(* Logix 5000 project; controller Sucrose_Main Emulate 5570 rev 20.12; software revision 20.01 *)

TASK _00_Master (continuous, watchdog 500 ms) : Master_Main
TASK _01_Sucrose (event, rate 10 ms, priority 10, watchdog 500 ms) : CIP_RemoteArea_AutoLogic, CIP_RemoteArea_EN2T_IO_Discrete_DO_E20_4, CIP_RemoteArea_EN2T_IO_Discrete_DO_E20_5, CIP_RemoteArea_EN2T_IO_Discrete_DO_E20_6, CIP_RemoteArea_EN2T_IO_Discrete_DO_E24_1, CIP_RemoteArea_EN2T_IO_Discrete_DO_E24_2, CIP_RemoteArea_EN2T_IO_Discrete_DO_E25_4, CIP_RemoteArea_EN2T_IO_Discrete_DO_E25_5, CIP_RemoteArea_EN2T_IO_Drives, DischargeArea_AutoLogic, DischargeArea_EN2T_IO_Discrete_DO_E20_3, DischargeArea_EN2T_IO_Discrete_DO_E20_4, DischargeArea_EN2T_IO_Discrete_DO_E20_5, DischargeArea_EN2T_IO_Discrete_DO_E20_6, DischargeArea_EN2T_IO_Discrete_DO_E20_7, DischargeArea_EN2T_IO_Discrete_DO_E24_3, DischargeArea_EN2T_IO_Drives, FiltrationArea_AutoLogic, FiltrationArea_EN2T_IO_Discrete_DO_E22_2, FiltrationArea_EN2T_IO_Discrete_DO_E22_3, FiltrationArea_EN2T_IO_Discrete_DO_E22_4

MODULES
   Local : Emulate 5570 (ICP 5, rev 20.12)
      EN2T_CCN : 1756-EN2T (ICP 1, Ethernet 192.168.15.49, rev 10.1)
      EN2T_IO : 1756-EN2T (ICP 2, Ethernet 192.168.1.1, rev 10.1)
         P620101 : PowerFlex 525-EENET (Ethernet 192.168.1.32, rev 3.1, Output RPI 20 ms)
         P230010 : PowerFlex 525-EENET (Ethernet 192.168.1.33, rev 4.1, Output RPI 20 ms)
         P230401 : PowerFlex 525-EENET (Ethernet 192.168.1.30, rev 2.2, Output RPI 20 ms)
         P230020 : PowerFlex 525-EENET (Ethernet 192.168.1.34, rev 4.1, Output RPI 20 ms)
         P230402 : PowerFlex 525-EENET (Ethernet 192.168.1.31, rev 4.1, Output RPI 20 ms)
         FLX_E25 : 1794-AENT (Ethernet 192.168.1.25, rev 4.1, Output RPI 20 ms)
            FLX_E25_2 : 1794-IB16 (Flex 2, rev 1.1)
            FLX_E25_5 : vendor 1 type 7 code 45 (Flex 5, rev 1.1)
            FLX_E25_4 : vendor 1 type 7 code 45 (Flex 4, rev 1.1)
            FLX_E25_3 : 1794-IB16 (Flex 3, rev 1.1)
            FLX_E25_1 : 1794-VHSC (Flex 1, rev 1.1, Output RPI 50 ms)
            FLX_E25_0 : vendor 1 type 10 code 25 (Flex 0, rev 2.1, Input RPI 80 ms)
         FLX_E20 : 1794-AENT (Ethernet 192.168.1.20, rev 4.1, Output RPI 20 ms)
            FLX_E20_7 : 1794-OW8 (Flex 7, rev 1.1)
            FLX_E20_4 : vendor 1 type 7 code 45 (Flex 4, rev 1.1)
            FLX_E20_5 : vendor 1 type 7 code 45 (Flex 5, rev 1.1)
            FLX_E20_1 : 1794-IB16 (Flex 1, rev 1.1)
            FLX_E20_6 : vendor 1 type 7 code 45 (Flex 6, rev 1.1)
            FLX_E20_2 : 1794-IB16 (Flex 2, rev 1.1)
            FLX_E20_0 : 1794-IB16 (Flex 0, rev 1.1)
            FLX_E20_3 : vendor 1 type 7 code 45 (Flex 3, rev 1.1)
         FLX_E24 : 1794-AENT (Ethernet 192.168.1.24, rev 4.1, Output RPI 20 ms)
            FLX_E24_5 : 1794-OW8 (Flex 5, rev 1.1)
            FLX_E24_0 : vendor 1 type 7 code 45 (Flex 0, rev 1.1)
            FLX_E24_4 : vendor 1 type 7 code 45 (Flex 4, rev 1.1)
            FLX_E24_1 : vendor 1 type 7 code 45 (Flex 1, rev 1.1)
            FLX_E24_2 : vendor 1 type 7 code 45 (Flex 2, rev 1.1)
            FLX_E24_3 : vendor 1 type 7 code 45 (Flex 3, rev 1.1)
            FLX_E24_6 : 1794-OW8 (Flex 6, rev 1.1)
         FLX_E21 : 1794-AENT (Ethernet 192.168.1.21, rev 4.1, Output RPI 20 ms)
            FLX_E21_1 : vendor 1 type 10 code 25 (Flex 1, rev 2.1, Input RPI 80 ms)
            FLX_E21_2 : vendor 1 type 10 code 25 (Flex 2, rev 2.1, Input RPI 80 ms)
            FLX_E21_0 : vendor 1 type 10 code 25 (Flex 0, rev 2.1, Input RPI 80 ms)
         FLX_E23 : 1794-AENT (Ethernet 192.168.1.23, rev 4.1, Output RPI 20 ms)
            FLX_E23_6 : 1794-IB16 (Flex 6, rev 1.1)
            FLX_E23_5 : 1794-IB16 (Flex 5, rev 1.1)
            FLX_E23_4 : 1794-IB16 (Flex 4, rev 1.1)
            FLX_E23_3 : 1794-IB16 (Flex 3, rev 1.1)
            FLX_E23_0 : vendor 1 type 10 code 25 (Flex 0, rev 2.1, Input RPI 80 ms)
            FLX_E23_2 : vendor 1 type 10 code 25 (Flex 2, rev 2.1, Input RPI 80 ms)
            FLX_E23_1 : vendor 1 type 10 code 25 (Flex 1, rev 2.1, Input RPI 80 ms)
         FLX_E22 : 1794-AENT (Ethernet 192.168.1.22, rev 4.1, Output RPI 20 ms)
            FLX_E22_2 : vendor 1 type 7 code 45 (Flex 2, rev 1.1)
            FLX_E22_7 : vendor 1 type 7 code 45 (Flex 7, rev 1.1)
            FLX_E22_5 : vendor 1 type 7 code 45 (Flex 5, rev 1.1)
            FLX_E22_1 : 1794-IB16 (Flex 1, rev 1.1)
            FLX_E22_4 : vendor 1 type 7 code 45 (Flex 4, rev 1.1)
            FLX_E22_0 : 1794-IB16 (Flex 0, rev 1.1)
            FLX_E22_3 : vendor 1 type 7 code 45 (Flex 3, rev 1.1)
            FLX_E22_6 : vendor 1 type 7 code 45 (Flex 6, rev 1.1)
END_MODULES

TYPE Area_Ladder :
STRUCT
   BIT_Comment : BOOL;   // For Rung Comment
   BIT_Alarm : DINT[1];   // For Logic Alarms
   BIT_ONS : BOOL[32];   // For Logic One Shot Bits
   TMR_Alarm : TIMER[25];   // For Logic Alarm Timers
   BIT_Logic : DINT[5];   // For Logic Bits
   SP_Logic : DINT[10];   // For Logic Setpoints
   TMR_Logic : TIMER[10];   // For Logic Timers
   CTR_Logic : COUNTER[5];   // For Logic Counters
   CALC_Logic : REAL[10];   // For Logic Math Calculations
   STRING_Logic : STRING[5];   // For Logic Strings
   BIT_HMI : DINT[10];   // For HMI Buttons
   SP_HMI : DINT[10];   // For HMI Setpoints
   STATUS_HMI : DINT[10];   // For HMI Display Words
   STATUS_BIT_HMI : DINT[10];   // For HMI Display Bits
   STRING_HMI : STRING[5];   // For HMI Strings
END_STRUCT
END_TYPE

TYPE Area_Program :
STRUCT
   BIT_Comment : BOOL;   // For Rung Comment
   BIT_Alarm : DINT[2];   // For Logic Alarms
   BIT_ONS : BOOL[128];   // For Logic One Shot Bits
   TMR_Alarm : TIMER[50];   // For Logic Alarm Timers
   BIT_Logic : DINT[10];   // For Logic Bits
   SP_Logic : DINT[25];   // For Logic Setpoints
   TMR_Logic : TIMER[50];   // For Logic Timers
   CTR_Logic : COUNTER[10];   // For Logic Counters
   CALC_Logic : REAL[25];   // For Logic Math Calculations
   STRING_Logic : STRING[5];   // For Logic Strings
   BIT_HMI : DINT[10];   // For HMI Buttons
   SP_HMI : DINT[25];   // For HMI Setpoints
   STATUS_HMI : DINT[10];   // For HMI Display Words
   STATUS_BIT_HMI : DINT[10];   // For HMI Display Bits
   STRING_HMI : STRING[5];   // For HMI Strings
   TMR_Debounce_On : TIMER[50];   // For Inputs Debounce Timer On
   TMR_Debounce_Off : TIMER[50];   // For Inputs Debounce Timer Off
END_STRUCT
END_TYPE

TYPE CIP_CURRENT_FUNCTIONS_REMOTE :
STRUCT
   F1 : DINT;   // CIP FUNCTION 1
   StepDescription : STRING;   // CIP STRING
   TIME : INT;   // CIP STEP TIME
   VALID : DINT;   // CIP VALID STEP CONFIRMATION
   F2 : DINT;   // CIP FUNCTION 1
   F3 : DINT;   // CIP FUNCTION 1
END_STRUCT
END_TYPE

TYPE CIP_MASTER_FUNCTIONS_REMOTE :
STRUCT
   F1 : DINT[130];   // CIP FUNCTION 1
   StepDescription : STRING[130];   // CIP STRING
   TIME : INT[130];   // CIP STEP TIME
   F2 : DINT[130];   // CIP FUNCTION 1
   F3 : DINT[130];   // CIP FUNCTION 1
END_STRUCT
END_TYPE

TYPE CIP_REMOTE :
STRUCT
   STEP : DINT;   // CIP STEP NUMBER
   STATES : CIP_STATES_REMOTE;
   STEP_TIMER : TIMER;   // CIP STEP TIMER
   CURRENT : CIP_CURRENT_FUNCTIONS_REMOTE;   // CIP CURRENT FUNCTIONS
   MASTER : CIP_MASTER_FUNCTIONS_REMOTE;   // CIP SETPOINTS
   BIT_ONS : BOOL[32];   // REMOTE ONE SHOTS
   Selected : BOOL;   // CIP CIRCUIT SELECTED
END_STRUCT
END_TYPE

TYPE CIP_STATES_REMOTE :
STRUCT
   RUNNING : BOOL;   // CIP RUNNING BIT
   PAUSED : BOOL;   // CIP PAUSED BIT
   HOLDING : BOOL;   // CIP HOLDING BIT
   COMPLETE : BOOL;   // CIP COMPLETE BIT
   STEP_DONE : BOOL;   // CIP STEP DONE BIT
   GOOD_MOVE : BOOL;   // CIP GOOD MOVE BIT
   VALID : DINT;   // CIP VALID STEP WORK
   TIMER_ENABLE : BOOL;   // CIP TIMER ENABLE
END_STRUCT
END_TYPE

TYPE Date_Time :
STRUCT
   Year : DINT;
   Month : DINT;
   Day : DINT;
   Hour : DINT;
   Minute : DINT;
   Second : DINT;
   Millisecond : DINT;
END_STRUCT
END_TYPE

TYPE User_Login :
STRUCT
   User_Data : STRING[20];
   Password_Data : STRING[20];
   User_Input : STRING;
   Password_Input : STRING;
   Password_Level : DINT;
   Current_User : STRING;
   Blank_User : STRING;
   Blank_Password : STRING;
   Default_User : STRING;
   Clear_User : BOOL;
   Logout_PB : BOOL;
   Good_User : BOOL;
   Login_PB : BOOL;
END_STRUCT
END_TYPE

ADD_ON_INSTRUCTION PF525_VFD_E_ENET   (* revision 2.0 Deluxe Edition, vendor Eric Casciaro *)
// QSI Typical Logic for VFD Controlled Motor
// Revision note:
// AOI Revisions After Multiple Startups:
// Added PID Execute Logic
// Added Manual On Reset Logic During Alarm
// Added Zone & Device Specific Alarm Ack Logic
// Added Zone & Device Specific Clear Fault Logic
// Added Zone Manual Mode Enable Logic
// Added Speed Display Units Option Logic
// Added Device Overspeed Option Logic
// Added HMI Popup Display Options Configuration
VAR_IN_OUT
   PF525_In : AB:PowerFlex525V_E_ED09CCB8:I:0; {required}
   PF525_Out : AB:PowerFlex525V_EENET_Drive:O:0; {required}
END_VAR
VAR_INPUT
   ALM_ACK : BOOL; {required}   // Zone Master Alarm Acknowledge
   MM_Enable : BOOL; {required}   // Zone Master Manual Mode Enable
   CLR_Fault : BOOL; {required}   // Zone Master Clear Fault Enable
   Config_TMR_On_Preset : DINT; {visible}   // Configure Delay Start Timer Preset
   Config_TMR_Off_Preset : DINT; {visible}   // Configure Delay Stop Timer Preset
   Config_TMR_Alm_Preset : DINT; {visible}   // Configure Device Alarm Timer Preset
   Config_MO_ALM_Reset : BOOL;   // Configure Whether .MO Bit Turns Off After Alarm Condition
END_VAR
VAR_OUTPUT
   Config_Drive_Overspeed : BOOL; {access Read Only}   // Configure Whether the Drive Max Speed is Oversped (0 = 100 % or 60 Hz) (1 = 200% or 120 Hz)
   Config_HMI_Units_SpeedFeedback : BOOL;   // Configure Whether Speed Feedback is Shown in % or Hertz (0=%) (1=Hz)
   Config_HMI_Control_Reverse : BOOL;   // Configure Whether HMI Popup Allows Reverse Control
   Config_HMI_Control_Jog : BOOL;   // Configure Whether HMI Popup Allows Jog Control
END_VAR
VAR_INPUT
   Config_AS1 : BOOL;   // Configure Usage of Auto Speed 1
   Config_AS2 : BOOL;   // Configure Usage of Auto Speed 2
   Config_AS3 : BOOL;   // Configure Usage of Auto Speed 3
   Config_AS4 : BOOL;   // Configure Usage of Auto Speed 4
   Config_AS5 : BOOL;   // Configure Usage of Auto Speed 5
   Config_PID : BOOL; {visible}   // Configure Usage of PID Loop
   Config_PID_Kp : REAL;   // Configure PID Proportional Gain
   Config_PID_Ki : REAL;   // Configure PID Integral Gain
   Config_PID_Kd : REAL;   // Configure PID Derivative Gain
   SP_AS1 : DINT;   // Auto Speed Setpoint
   SP_AS2 : DINT;   // Auto Speed #2 Setpoint
   SP_AS3 : DINT;   // Auto Speed #2 Setpoint
   SP_AS4 : DINT;   // Auto Speed #2 Setpoint
   SP_AS5 : DINT;   // Auto Speed #2 Setpoint
   SP_PID_PV : REAL;   // PID Process Variable
   SP_PID_SP : REAL;   // PID Set Point
   SP_PID_SO : REAL;   // PID Set Output (0-100%) (0-200% If Drive Needs Overspeed)
   AS1_Enable : BOOL;   // Auto Speed 1 Enable From Logic
   AS2_Enable : BOOL;   // Auto Speed 2 Enable From Logic
   AS3_Enable : BOOL;   // Auto Speed 3 Enable From Logic
   AS4_Enable : BOOL;   // Auto Speed 4 Enable From Logic
   AS5_Enable : BOOL;   // Auto Speed 5 Enable From Logic
   PID_Enable : BOOL;   // Pid Loop Enable From Logic
   PID_SWM_Enable : BOOL;   // PID Software Manual Enable From Logic
   Start_Permissive : BOOL;   // Drive Start Run Permissive From Logic (EStop Ok, Disconnect Ok, Drive Enabled, Safe Off Ok)
   Reverse_Enable : BOOL;   // Drive Reverse Command From Logic
   HMI_MM : BOOL; {visible}   // Manual Mode Bit
   HMI_MO : BOOL; {visible}   // Manual On Bit
   HMI_MS : DINT; {visible}   // Manual Speed Setpoint
   HMI_SP_PID_SO : REAL;   // HMI PID Set Output (0-100%) (0-200% If Drive Needs Overspeed)
   HMI_ALM_ACK : BOOL;   // AOI Device Alarm Acknowledge
   HMI_CLR_Fault : BOOL;   // AOI Device Clear Fault
   HMI_PID_SWM : BOOL;   // HMI PID Loop .SWM Mode Selected
END_VAR
VAR_OUTPUT
   Started : BOOL; {visible}   // Drive Started Status
   Running : BOOL; {visible}   // Drive Started Status
   HMI_CommandSpeed : DINT; {visible}   // Commanded Frequency Status
   HMI_FeedbackSpeed : DINT; {visible}   // Feedback Frequency Status
   ALM : BOOL; {visible}   // Drive & Motor Combined Alarm Bit
   PID_Enabled : BOOL;   // PID Loop Enabled Status
   PID_CV : REAL;   // PID Control Variable
   PID_Out : REAL;   // PID Output Status
   PID_PVMax : DINT;   // PID Process Variable Max Status
END_VAR
VAR
   ONS : BOOL[32]; {access None}
   TMR_Off : TIMER; {access None}   // Device Output Timer On
   TMR_On : TIMER; {access None}   // Device Output Timer Off
   TMR_Alm : TIMER; {access None}   // Device Alarm Timer
   BIT_Comment : BOOL; {access None}
   PID_En : BOOL; {access None}   // PID Loop Enabled
   PID : PID := (CTL := 2097152, NOBC := 1, MAXO := 100.0, UPD := 0.1, MAXCV := 1200.0); {access None}   // Device PID Loop
   PID_TMR_On : TIMER := (PRE := 500); {access None}   // PID Execute Timer (Should Be 5 x PV Update Rate)
END_VAR

ROUTINE Logic   (* ladder *)
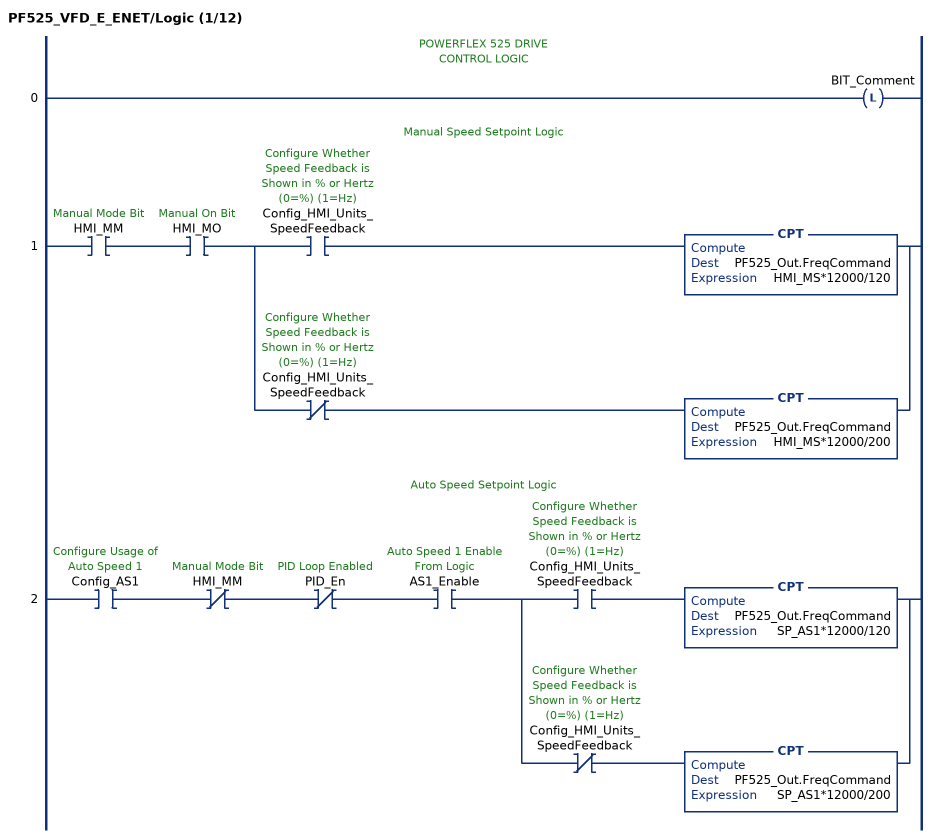
   // POWERFLEX 525 DRIVE
   // CONTROL LOGIC
   0: OTL(BIT_Comment);
   // Manual Speed Setpoint Logic
   1: XIC(HMI_MM)XIC(HMI_MO)[XIC(Config_HMI_Units_SpeedFeedback) CPT(PF525_Out.FreqCommand,HMI_MS*12000/120) ,XIO(Config_HMI_Units_SpeedFeedback) CPT(PF525_Out.FreqCommand,HMI_MS*12000/200) ];
   // Auto Speed Setpoint Logic
   2: XIC(Config_AS1)XIO(HMI_MM)XIO(PID_En)XIC(AS1_Enable)[XIC(Config_HMI_Units_SpeedFeedback) CPT(PF525_Out.FreqCommand,SP_AS1*12000/120) ,XIO(Config_HMI_Units_SpeedFeedback) CPT(PF525_Out.FreqCommand,SP_AS1*12000/200) ];
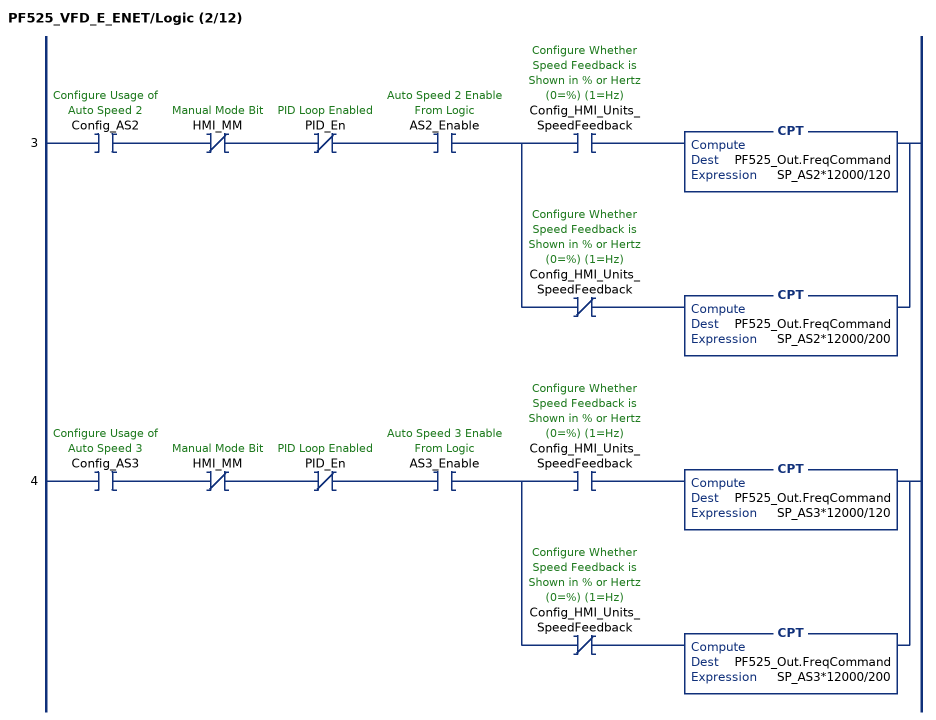
   3: XIC(Config_AS2)XIO(HMI_MM)XIO(PID_En)XIC(AS2_Enable)[XIC(Config_HMI_Units_SpeedFeedback) CPT(PF525_Out.FreqCommand,SP_AS2*12000/120) ,XIO(Config_HMI_Units_SpeedFeedback) CPT(PF525_Out.FreqCommand,SP_AS2*12000/200) ];
   4: XIC(Config_AS3)XIO(HMI_MM)XIO(PID_En)XIC(AS3_Enable)[XIC(Config_HMI_Units_SpeedFeedback) CPT(PF525_Out.FreqCommand,SP_AS3*12000/120) ,XIO(Config_HMI_Units_SpeedFeedback) CPT(PF525_Out.FreqCommand,SP_AS3*12000/200) ];
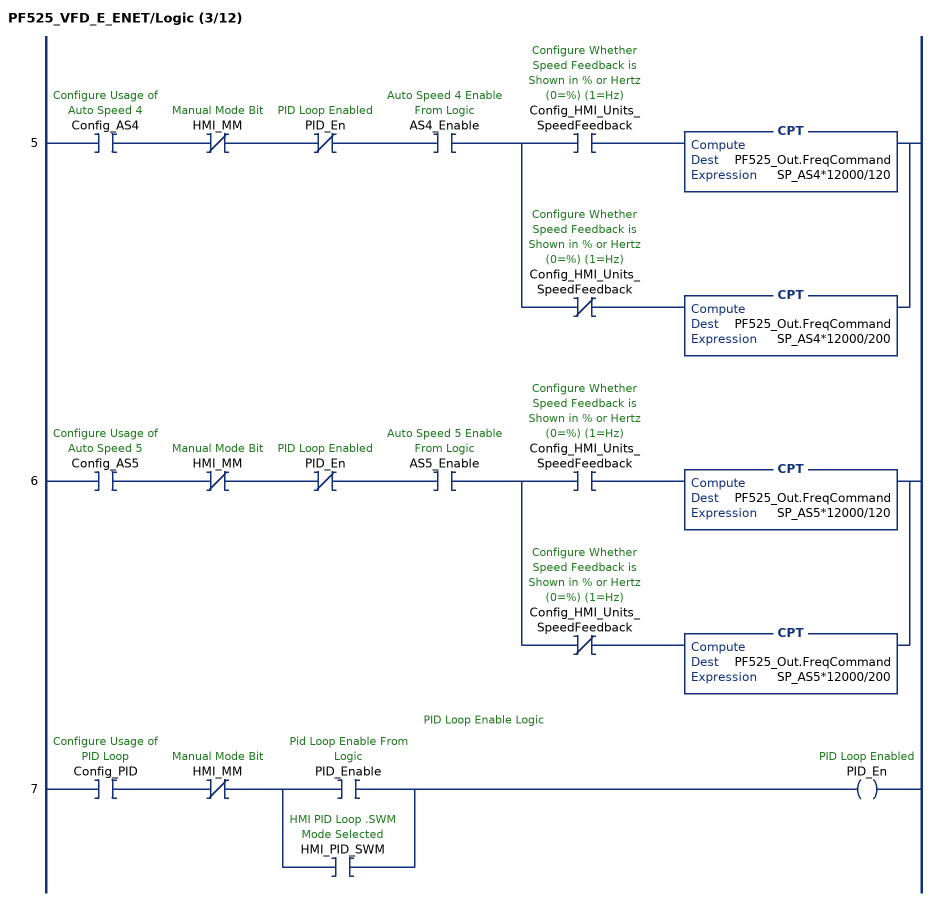
   5: XIC(Config_AS4)XIO(HMI_MM)XIO(PID_En)XIC(AS4_Enable)[XIC(Config_HMI_Units_SpeedFeedback) CPT(PF525_Out.FreqCommand,SP_AS4*12000/120) ,XIO(Config_HMI_Units_SpeedFeedback) CPT(PF525_Out.FreqCommand,SP_AS4*12000/200) ];
   6: XIC(Config_AS5)XIO(HMI_MM)XIO(PID_En)XIC(AS5_Enable)[XIC(Config_HMI_Units_SpeedFeedback) CPT(PF525_Out.FreqCommand,SP_AS5*12000/120) ,XIO(Config_HMI_Units_SpeedFeedback) CPT(PF525_Out.FreqCommand,SP_AS5*12000/200) ];
   // PID Loop Enable Logic
   7: XIC(Config_PID)XIO(HMI_MM)[XIC(PID_Enable) ,XIC(HMI_PID_SWM) ]OTE(PID_En);
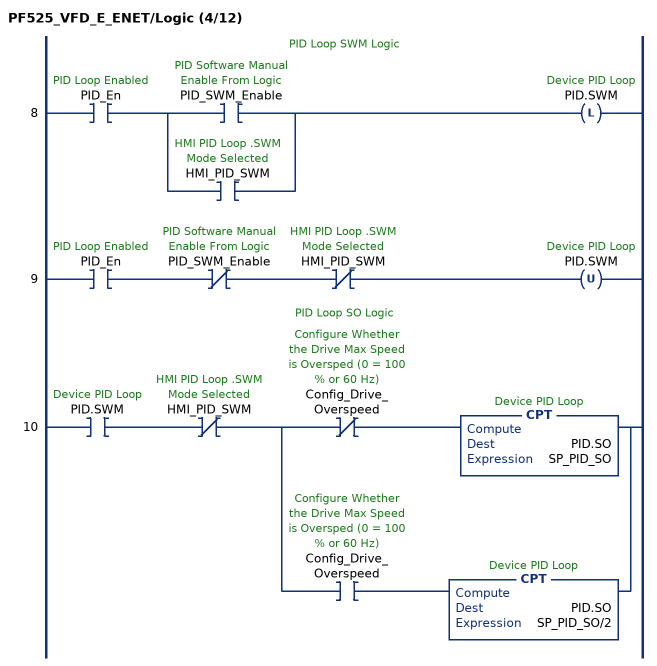
   // PID Loop SWM Logic
   8: XIC(PID_En)[XIC(PID_SWM_Enable) ,XIC(HMI_PID_SWM) ]OTL(PID.SWM);
   9: XIC(PID_En)XIO(PID_SWM_Enable)XIO(HMI_PID_SWM)OTU(PID.SWM);
   // PID Loop SO Logic
   10: XIC(PID.SWM)XIO(HMI_PID_SWM)[XIO(Config_Drive_Overspeed) CPT(PID.SO,SP_PID_SO) ,XIC(Config_Drive_Overspeed) CPT(PID.SO,SP_PID_SO/2) ];
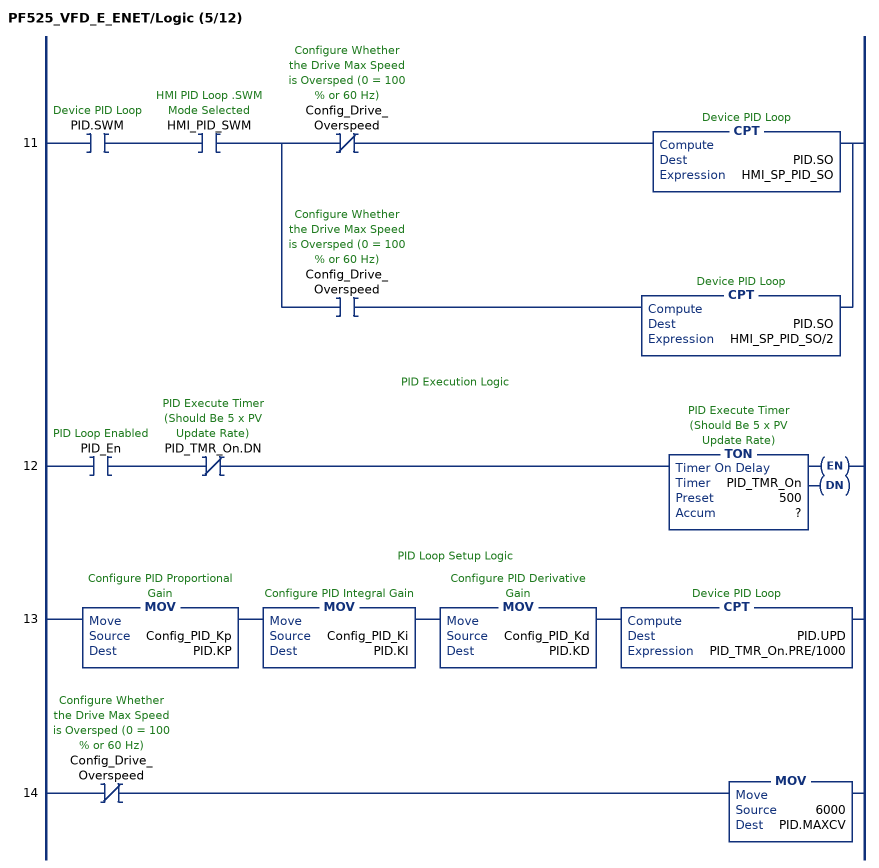
   11: XIC(PID.SWM)XIC(HMI_PID_SWM)[XIO(Config_Drive_Overspeed) CPT(PID.SO,HMI_SP_PID_SO) ,XIC(Config_Drive_Overspeed) CPT(PID.SO,HMI_SP_PID_SO/2) ];
   // PID Execution Logic
   12: XIC(PID_En)XIO(PID_TMR_On.DN)TON(PID_TMR_On,?,?);
   // PID Loop Setup Logic
   13: MOV(Config_PID_Kp,PID.KP)MOV(Config_PID_Ki,PID.KI)MOV(Config_PID_Kd,PID.KD)CPT(PID.UPD,PID_TMR_On.PRE/1000);
   14: XIO(Config_Drive_Overspeed)MOV(6000,PID.MAXCV);
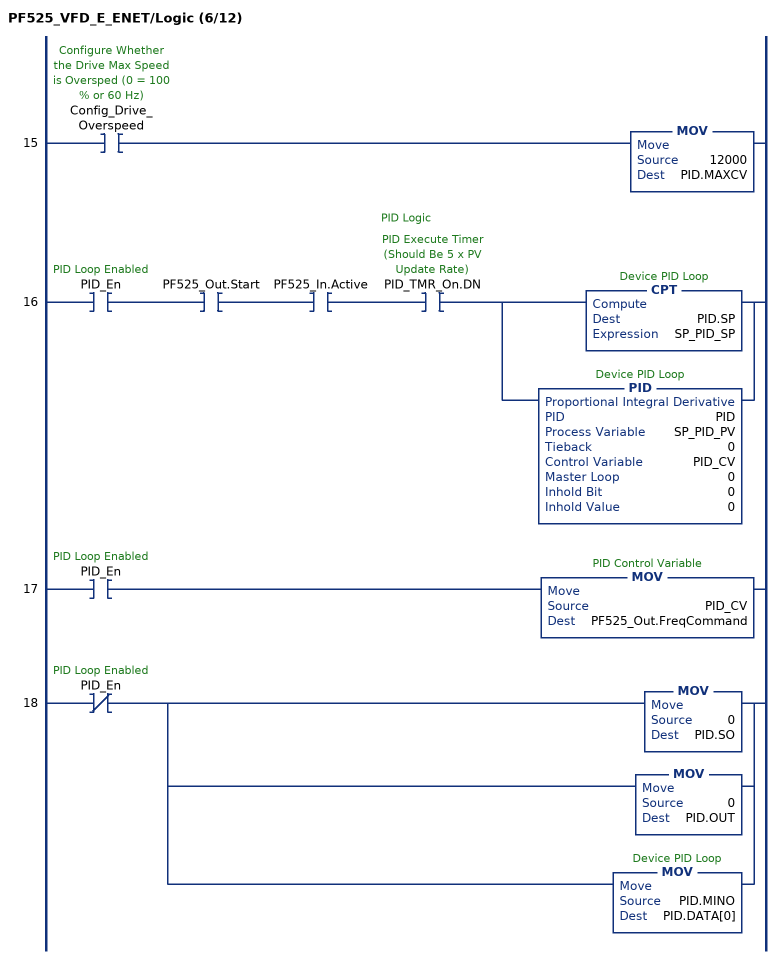
   15: XIC(Config_Drive_Overspeed)MOV(12000,PID.MAXCV);
   // PID Logic
   16: XIC(PID_En)XIC(PF525_Out.Start)XIC(PF525_In.Active)XIC(PID_TMR_On.DN)[CPT(PID.SP,SP_PID_SP) ,PID(PID,SP_PID_PV,0,PID_CV,0,0,0) ];
   17: XIC(PID_En)MOV(PID_CV,PF525_Out.FreqCommand);
   18: XIO(PID_En)[MOV(0,PID.SO) ,MOV(0,PID.OUT) ,MOV(PID.MINO,PID.DATA[0]) ];
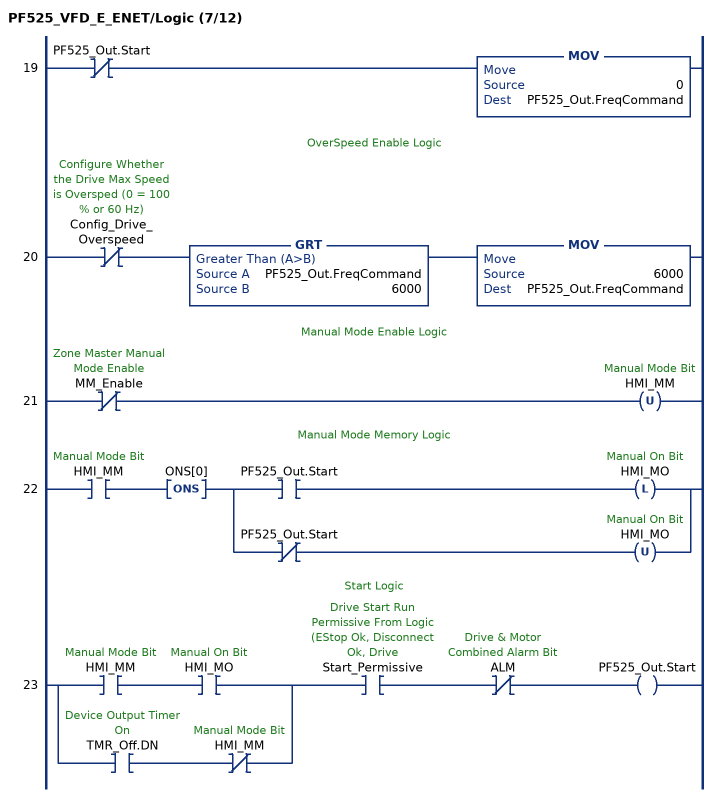
   19: XIO(PF525_Out.Start)MOV(0,PF525_Out.FreqCommand);
   // OverSpeed Enable Logic
   20: XIO(Config_Drive_Overspeed)GRT(PF525_Out.FreqCommand,6000)MOV(6000,PF525_Out.FreqCommand);
   // Manual Mode Enable Logic
   21: XIO(MM_Enable)OTU(HMI_MM);
   // Manual Mode Memory Logic
   22: XIC(HMI_MM)ONS(ONS[0])[XIC(PF525_Out.Start) OTL(HMI_MO) ,XIO(PF525_Out.Start) OTU(HMI_MO) ];
   // Start Logic
   23: [XIC(HMI_MM) XIC(HMI_MO) ,XIC(TMR_Off.DN) XIO(HMI_MM) ]XIC(Start_Permissive)XIO(ALM)OTE(PF525_Out.Start);
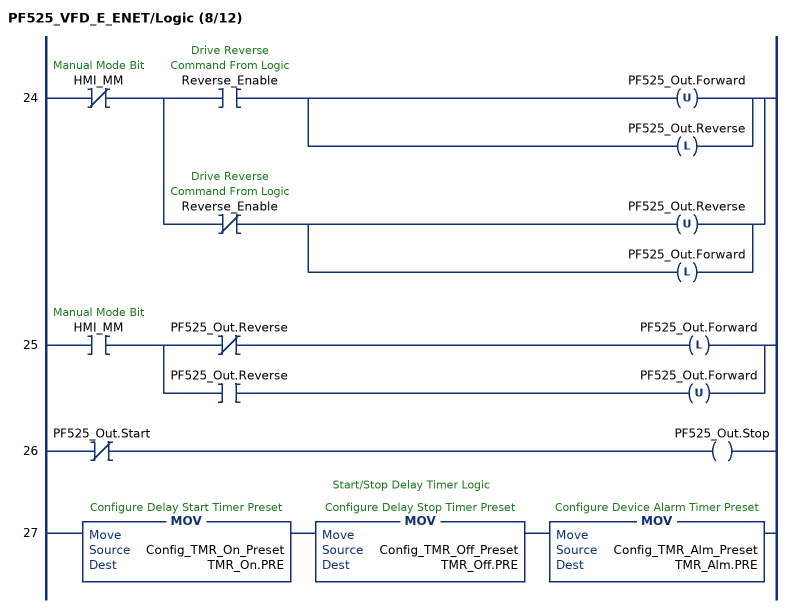
   24: XIO(HMI_MM)[XIC(Reverse_Enable) [OTU(PF525_Out.Forward) ,OTL(PF525_Out.Reverse) ] ,XIO(Reverse_Enable) [OTU(PF525_Out.Reverse) ,OTL(PF525_Out.Forward) ] ];
   25: XIC(HMI_MM)[XIO(PF525_Out.Reverse) OTL(PF525_Out.Forward) ,XIC(PF525_Out.Reverse) OTU(PF525_Out.Forward) ];
   26: XIO(PF525_Out.Start)OTE(PF525_Out.Stop);
   // Start/Stop Delay Timer Logic
   27: MOV(Config_TMR_On_Preset,TMR_On.PRE)MOV(Config_TMR_Off_Preset,TMR_Off.PRE)MOV(Config_TMR_Alm_Preset,TMR_Alm.PRE);
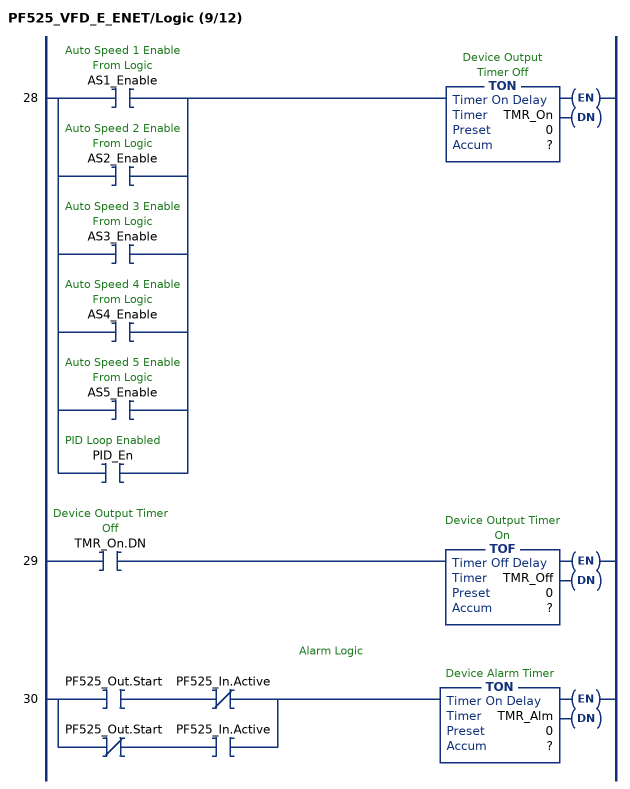
   28: [XIC(AS1_Enable) ,XIC(AS2_Enable) ,XIC(AS3_Enable) ,XIC(AS4_Enable) ,XIC(AS5_Enable) ,XIC(PID_En) ]TON(TMR_On,?,?);
   29: XIC(TMR_On.DN)TOF(TMR_Off,?,?);
   // Alarm Logic
   30: [XIC(PF525_Out.Start) XIO(PF525_In.Active) ,XIO(PF525_Out.Start) XIC(PF525_In.Active) ]TON(TMR_Alm,?,?);
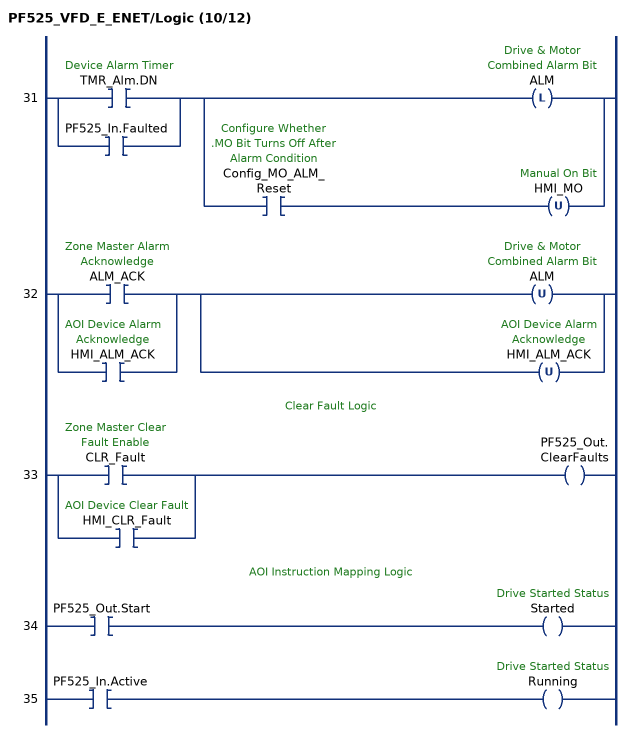
   31: [XIC(TMR_Alm.DN) ,XIC(PF525_In.Faulted) ][OTL(ALM) ,XIC(Config_MO_ALM_Reset) OTU(HMI_MO) ];
   32: [XIC(ALM_ACK) ,XIC(HMI_ALM_ACK) ][OTU(ALM) ,OTU(HMI_ALM_ACK) ];
   // Clear Fault Logic
   33: [XIC(CLR_Fault) ,XIC(HMI_CLR_Fault) ]OTE(PF525_Out.ClearFaults);
   // AOI Instruction Mapping Logic
   34: XIC(PF525_Out.Start)OTE(Started);
   35: XIC(PF525_In.Active)OTE(Running);
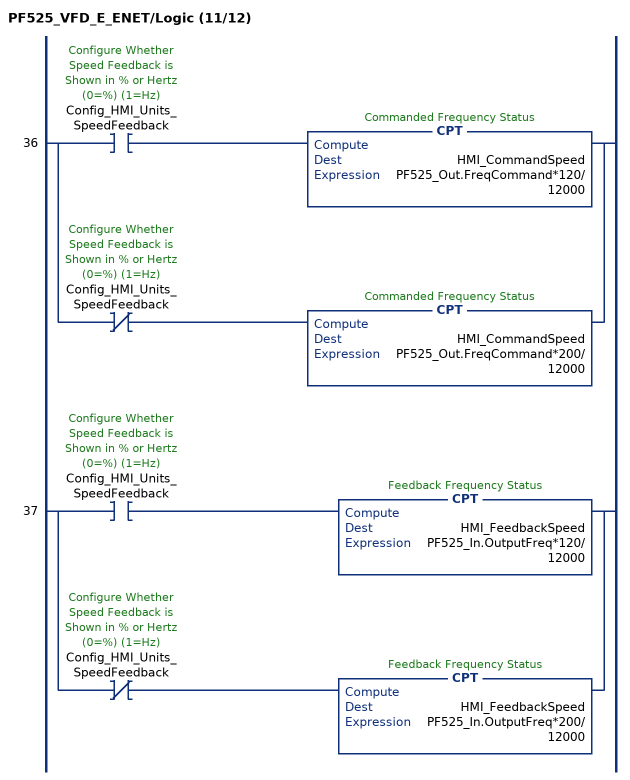
   36: [XIC(Config_HMI_Units_SpeedFeedback) CPT(HMI_CommandSpeed,PF525_Out.FreqCommand*120/12000) ,XIO(Config_HMI_Units_SpeedFeedback) CPT(HMI_CommandSpeed,PF525_Out.FreqCommand*200/12000) ];
   37: [XIC(Config_HMI_Units_SpeedFeedback) CPT(HMI_FeedbackSpeed,PF525_In.OutputFreq*120/12000) ,XIO(Config_HMI_Units_SpeedFeedback) CPT(HMI_FeedbackSpeed,PF525_In.OutputFreq*200/12000) ];
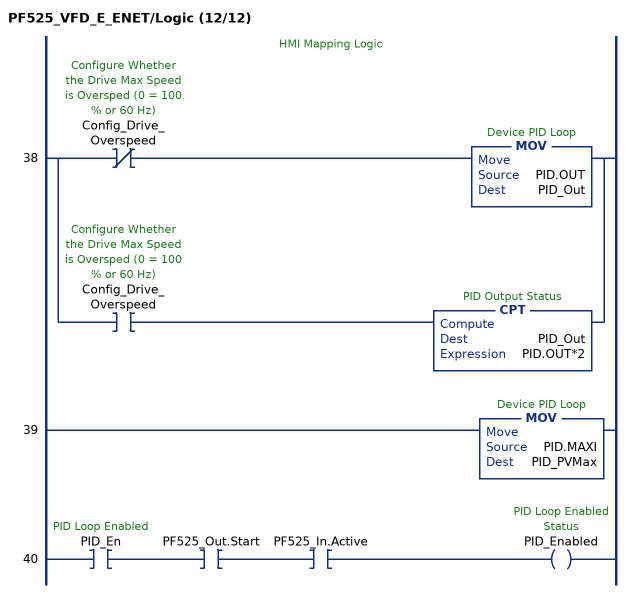
   // HMI Mapping Logic
   38: [XIO(Config_Drive_Overspeed) MOV(PID.OUT,PID_Out) ,XIC(Config_Drive_Overspeed) CPT(PID_Out,PID.OUT*2) ];
   39: MOV(PID.MAXI,PID_PVMax);
   40: XIC(PID_En)XIC(PF525_Out.Start)XIC(PF525_In.Active)OTE(PID_Enabled);
END_ROUTINE
END_ADD_ON_INSTRUCTION

ADD_ON_INSTRUCTION QSI_Analog_Valve   (* revision 2.0 *)
// Revision note:
// Added Feedback Out of Range Alarm
// Added Config Param to select Analog Feedback
// Added Config Param to select N.O. or N.C. Valve
// Added Manual On Reset Logic During Alarm
// Added Zone & Device Specific Alarm Ack Logic
// Added Zone Manual Mode Enable Logic
VAR_OUTPUT
   DO_Energize : BOOL; {access Read Only, required}   // Alias to OutputCard to Energize Discrete Output
   AO_CommandPosition : REAL; {access Read Only, required}   // Alias to AO Tag to Control Analog Output
END_VAR
VAR_INPUT
   AI_Position_Feedback : REAL; {required}   // Alias to AI Tag to Confirm Device is at Desired Position Note: Must be scaled to value of Config_Analog_PositionMaxScaled
   PID_ProcessVariable : REAL; {required}   // Alias to AI Tag that Will Serve as PID Loop Process Variable
   ALM_ACK : BOOL; {required}   // Alias to Zone Master Alarm Acknowledge
   MM_Enable : BOOL; {required}   // Alias to Zone Master Manual Mode Enable
   Config_NO_Valve : BOOL; {visible}   // Configure Whether Valve is Normally Closed (0 = N.C., 1 = N.O.)
   Config_Position_Feedback : BOOL; {visible}   // Config Whether Device has Position Feedback (0= No, 1= Yes) Note: Alarm Disabled if No Feedback
   Config_MO_ResetOnAlarm : BOOL := 1; {visible}   // Configure Whether .MO Bit Turns Off when Device Alarm Condition Exists
   Config_AO_PositionMaxRaw : REAL := 30840.0; {visible}   // Configure Analog Card Max Raw Analog Value
   Config_Analog_PositionMaxScaled : REAL := 100.0; {visible}   // Configure Analog Device Max Scaled Value
   Config_TMR_Alm_Preset_ms : DINT; {visible}   // Configure Device AlarmTimer Preset In Milliseconds
   Config_TMR_Off_Preset_ms : DINT; {visible}   // Configure Delay Stop Timer Preset In Milliseconds
   Config_TMR_On_Preset_ms : DINT; {visible}   // Configure Delay Start Timer Preset In Milliseconds
   Config_PID : BOOL; {visible}   // Configure Usage of PID Loop
END_VAR
VAR_OUTPUT
   HMI_PID_Enabled : BOOL; {access Read Only, visible}   // PID Loop Enabled To HMI
   HMI_PID_SP : REAL; {visible}   // PID SP to HMI
   HMI_PID_PV : REAL; {visible}   // PID PV to HMI
   HMI_PID_Out : REAL; {access Read Only, visible}   // PID Output to HMI
END_VAR
VAR_INPUT
   HMI_MM : BOOL; {visible}   // Manual Mode Bit
   HMI_MO : BOOL; {visible}   // Manual On Bit
   HMI_MS : DINT; {visible}   // Manual Position Setpoint
END_VAR
VAR_OUTPUT
   HMI_CommandedPosition : REAL; {visible}   // Device Commanded Position to HMI
   HMI_FeedbackPosition : REAL; {visible}   // Device Feedback Position to HMI
END_VAR
VAR_INPUT
   HMI_ALM_ACK : BOOL;   // AOI Device Specific Alarm Acknowledge From HMI
END_VAR
VAR_OUTPUT
   HMI_Alarmed : BOOL;   // Alarm Status To HMI
   HMI_Opened : BOOL;   // Opened Status To HMI
   HMI_Closed : BOOL;   // Closed Status To HMI
END_VAR
VAR_INPUT
   HMI_PID_SWM : BOOL;   // HMI PID Loop .SWM Mode Selected
   HMI_SP_PID_SO : REAL;   // HMI PID Set Output (0-100%) (0-200% If Drive Needs Overspeed)
   HMI_PID_Kp : REAL;
   HMI_PID_Ki : REAL;
   HMI_PID_Kd : REAL;
END_VAR
VAR_OUTPUT
   HMI_PID_PVMax : DINT;   // PID Process Variable Max Status
END_VAR
VAR_INPUT
   SP_AS1 : DINT;   // Auto Position #1 Setpoint
   SP_AS2 : DINT;   // Auto Position #2 Setpoint
   SP_AS3 : DINT;   // Auto Position #3 Setpoint
   SP_AS4 : DINT;   // Auto Position #4 Setpoint
   SP_AS5 : DINT;   // Auto Position #5 Setpoint
   SP_PID_SP : REAL;   // Setpoint for Desired Setpoint of PID Process Variable
   SP_PID_SO : REAL;   // Setpoint for PID Manual Set Output Position
   Energize_Permissive : BOOL;   // Valve Permissive From Logic (EStop Ok)
   AS1_Enable : BOOL;   // Auto Setpoint 1 Enable Interlock From Logic
   AS2_Enable : BOOL;   // Auto Setpoint 2 Enable Interlock From Logic
   AS3_Enable : BOOL;   // Auto Setpoint 3 Enable Interlock From Logic
   AS4_Enable : BOOL;   // Auto Setpoint 4 Enable Interlock From Logic
   AS5_Enable : BOOL;   // Auto Setpoint 5 Enable Interlock From Logic
   PID_Enable : BOOL;   // PID Enable Interlock From Logic
   PID_SWM_Enable : BOOL;   // PID.SWM Enable Interlock From Logic
END_VAR
VAR_OUTPUT
   ALM : BOOL; {visible}   // Device Alarm
END_VAR
VAR_INPUT
   Comment : BOOL;   // Comment for Description Rung to Start Each Routine
   Unused_Input_BOOL : BOOL;   // Trash Tag For Required AOI Input Variables That Are Unused for Current Device (Type Boolean)
END_VAR
VAR_OUTPUT
   Unused_Output_BOOL : BOOL;   // Trash Tag For Required AOI Output Variables That Are Unused for Current Device (Type Boolean)
END_VAR
VAR_INPUT
   Unused_Input_Analog : REAL;   // Trash Tag For Required AOI Input Variables That Are Unused for Current Device (Type Analog)
END_VAR
VAR_OUTPUT
   Unused_Output_Analog : REAL;   // Trash Tag For Required AOI Output Variables That Are Unused for Current Device (Type Analog)
END_VAR
VAR
   ONS : BOOL[32];
   PID_En : BOOL;   // PID Loop Enabled
   PID : PID := (CTL := 35651584, CA := 1, NOBC := 1, UPD := 0.01, MAXCV := 30840.0);
   PID_TMR_On : TIMER := (PRE := 500); {access None}   // PID Execute Timer (Should Be 5 x PV Update Rate)
   TMR_On : TIMER; {access None}
   TMR_Off : TIMER; {access None}
   TMR_Alm : TIMER; {access None}
   Position_Alm_UpperLimit : REAL; {access None}
   Position_Alm_LowerLimit : REAL; {access None}
   PID_CV : DINT; {access None}
   Position_UpperLimit : REAL; {access None}
   Position_LowerLimit : REAL; {access None}
END_VAR

ROUTINE Logic   (* ladder *)
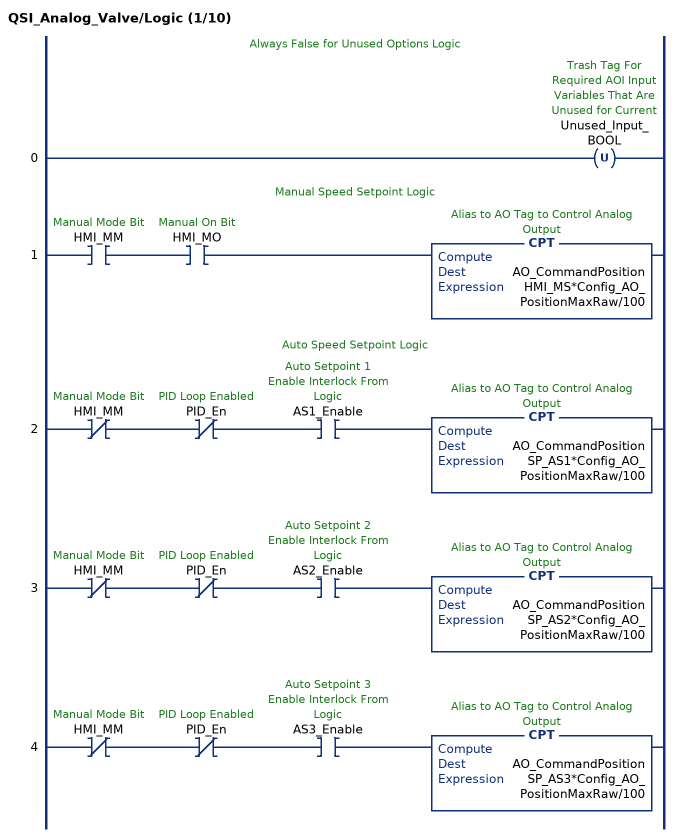
   // Always False for Unused Options Logic
   0: OTU(Unused_Input_BOOL);
   // Manual Speed Setpoint Logic
   1: XIC(HMI_MM)XIC(HMI_MO)CPT(AO_CommandPosition,HMI_MS*Config_AO_PositionMaxRaw/100);
   // Auto Speed Setpoint Logic
   2: XIO(HMI_MM)XIO(PID_En)XIC(AS1_Enable)CPT(AO_CommandPosition,SP_AS1*Config_AO_PositionMaxRaw/100);
   3: XIO(HMI_MM)XIO(PID_En)XIC(AS2_Enable)CPT(AO_CommandPosition,SP_AS2*Config_AO_PositionMaxRaw/100);
   4: XIO(HMI_MM)XIO(PID_En)XIC(AS3_Enable)CPT(AO_CommandPosition,SP_AS3*Config_AO_PositionMaxRaw/100);
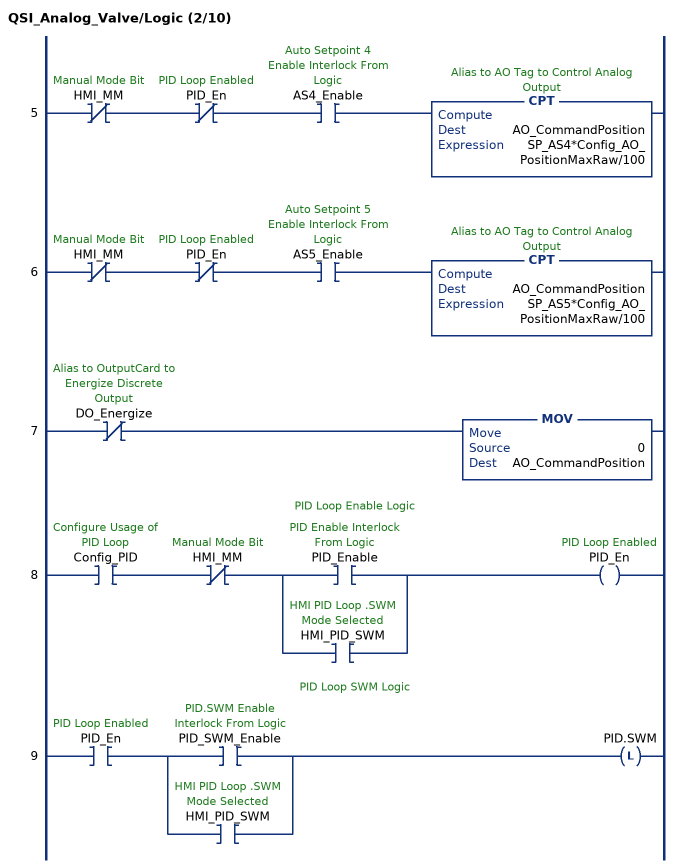
   5: XIO(HMI_MM)XIO(PID_En)XIC(AS4_Enable)CPT(AO_CommandPosition,SP_AS4*Config_AO_PositionMaxRaw/100);
   6: XIO(HMI_MM)XIO(PID_En)XIC(AS5_Enable)CPT(AO_CommandPosition,SP_AS5*Config_AO_PositionMaxRaw/100);
   7: XIO(DO_Energize)MOV(0,AO_CommandPosition);
   // PID Loop Enable Logic
   8: XIC(Config_PID)XIO(HMI_MM)[XIC(PID_Enable) ,XIC(HMI_PID_SWM) ]OTE(PID_En);
   // PID Loop SWM Logic
   9: XIC(PID_En)[XIC(PID_SWM_Enable) ,XIC(HMI_PID_SWM) ]OTL(PID.SWM);
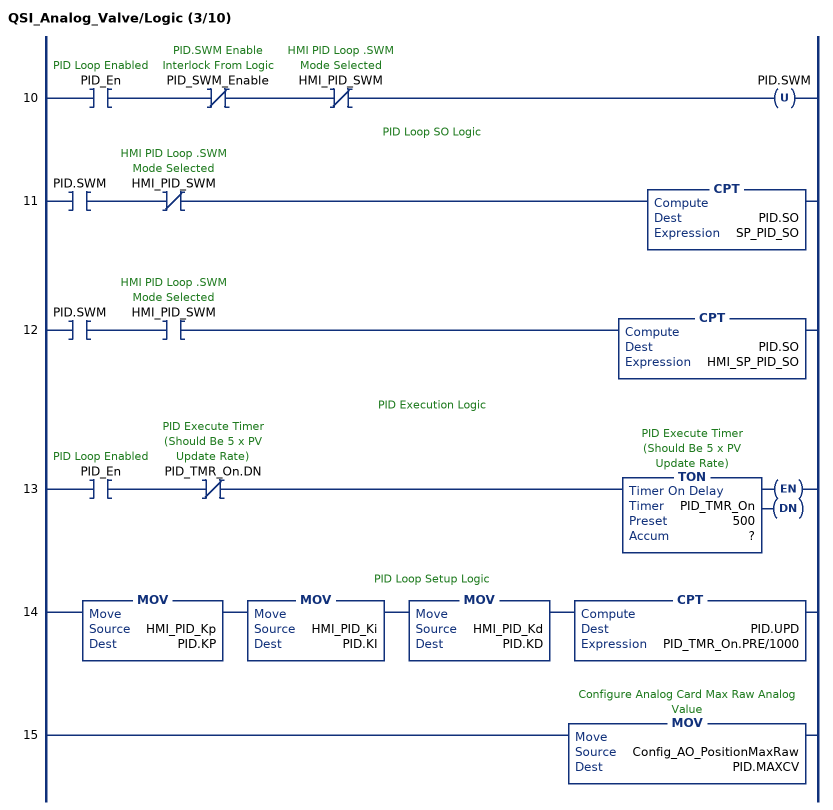
   10: XIC(PID_En)XIO(PID_SWM_Enable)XIO(HMI_PID_SWM)OTU(PID.SWM);
   // PID Loop SO Logic
   11: XIC(PID.SWM)XIO(HMI_PID_SWM)CPT(PID.SO,SP_PID_SO);
   12: XIC(PID.SWM)XIC(HMI_PID_SWM)CPT(PID.SO,HMI_SP_PID_SO);
   // PID Execution Logic
   13: XIC(PID_En)XIO(PID_TMR_On.DN)TON(PID_TMR_On,?,?);
   // PID Loop Setup Logic
   14: MOV(HMI_PID_Kp,PID.KP)MOV(HMI_PID_Ki,PID.KI)MOV(HMI_PID_Kd,PID.KD)CPT(PID.UPD,PID_TMR_On.PRE/1000);
   15: MOV(Config_AO_PositionMaxRaw,PID.MAXCV);
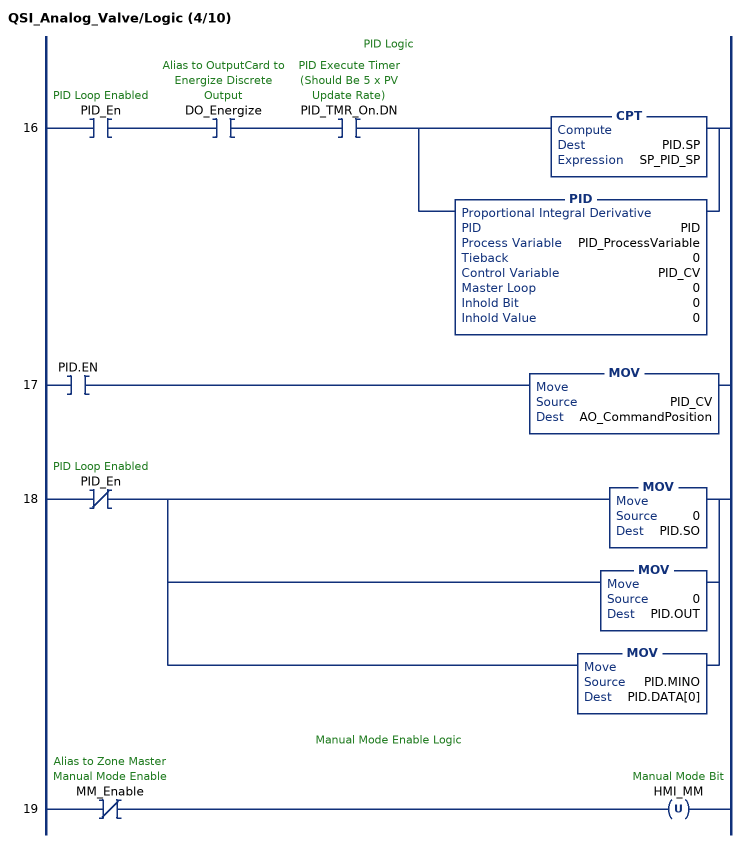
   // PID Logic
   16: XIC(PID_En)XIC(DO_Energize)XIC(PID_TMR_On.DN)[CPT(PID.SP,SP_PID_SP) ,PID(PID,PID_ProcessVariable,0,PID_CV,0,0,0) ];
   17: XIC(PID.EN)MOV(PID_CV,AO_CommandPosition);
   18: XIO(PID_En)[MOV(0,PID.SO) ,MOV(0,PID.OUT) ,MOV(PID.MINO,PID.DATA[0]) ];
   // Manual Mode Enable Logic
   19: XIO(MM_Enable)OTU(HMI_MM);
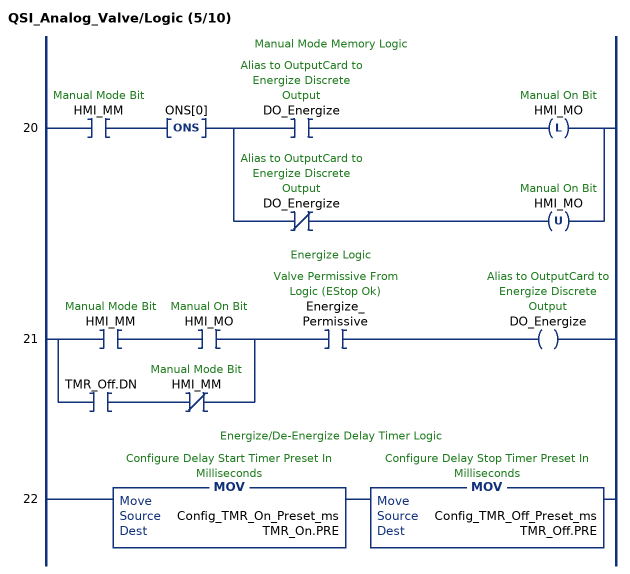
   // Manual Mode Memory Logic
   20: XIC(HMI_MM)ONS(ONS[0])[XIC(DO_Energize) OTL(HMI_MO) ,XIO(DO_Energize) OTU(HMI_MO) ];
   // Energize Logic
   21: [XIC(HMI_MM) XIC(HMI_MO) ,XIC(TMR_Off.DN) XIO(HMI_MM) ]XIC(Energize_Permissive)OTE(DO_Energize);
   // Energize/De-Energize Delay Timer Logic
   22: MOV(Config_TMR_On_Preset_ms,TMR_On.PRE)MOV(Config_TMR_Off_Preset_ms,TMR_Off.PRE);
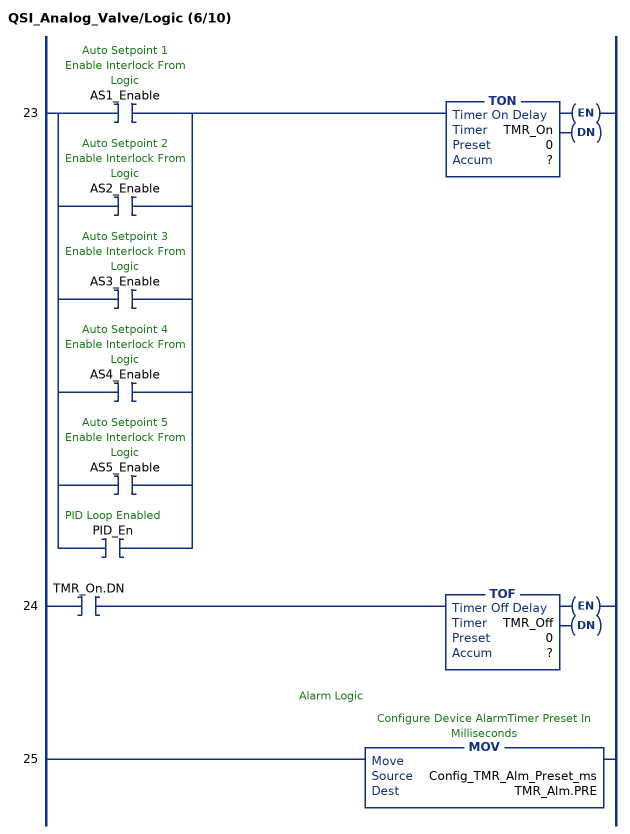
   23: [XIC(AS1_Enable) ,XIC(AS2_Enable) ,XIC(AS3_Enable) ,XIC(AS4_Enable) ,XIC(AS5_Enable) ,XIC(PID_En) ]TON(TMR_On,?,?);
   24: XIC(TMR_On.DN)TOF(TMR_Off,?,?);
   // Alarm Logic
   25: MOV(Config_TMR_Alm_Preset_ms,TMR_Alm.PRE);
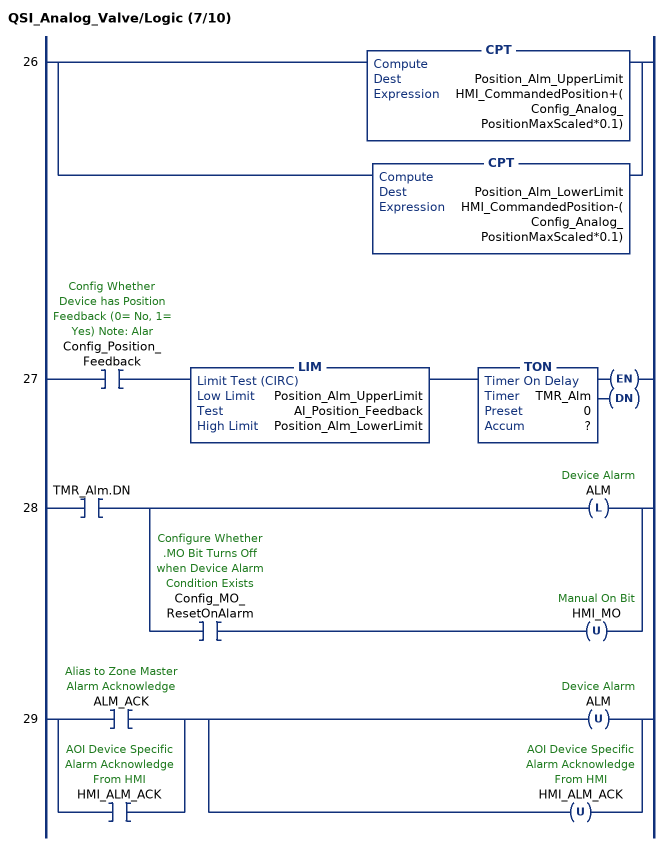
   26: [CPT(Position_Alm_UpperLimit,HMI_CommandedPosition+(Config_Analog_PositionMaxScaled*0.1)) ,CPT(Position_Alm_LowerLimit,HMI_CommandedPosition-(Config_Analog_PositionMaxScaled*0.1)) ];
   27: XIC(Config_Position_Feedback)LIM(Position_Alm_UpperLimit,AI_Position_Feedback,Position_Alm_LowerLimit)TON(TMR_Alm,?,?);
   28: XIC(TMR_Alm.DN)[OTL(ALM) ,XIC(Config_MO_ResetOnAlarm) OTU(HMI_MO) ];
   29: [XIC(ALM_ACK) ,XIC(HMI_ALM_ACK) ][OTU(ALM) ,OTU(HMI_ALM_ACK) ];
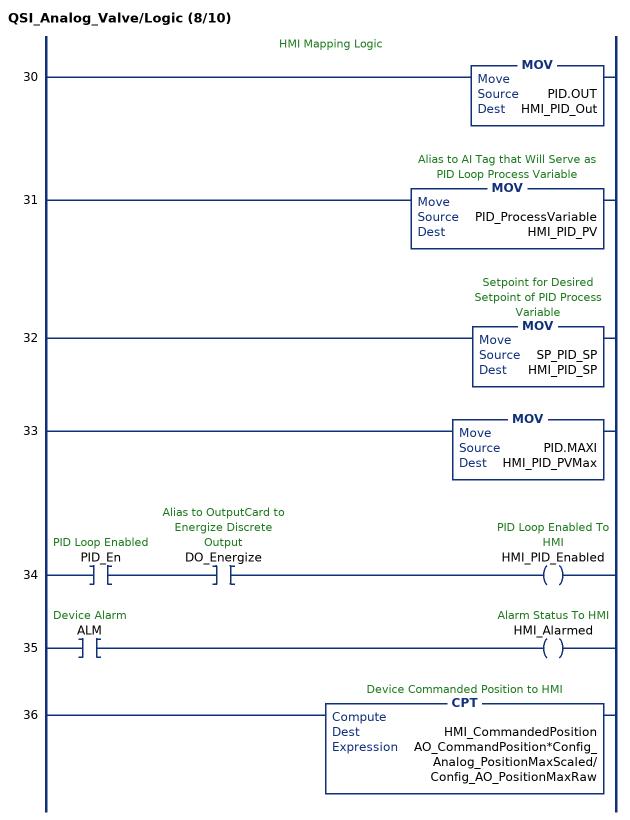
   // HMI Mapping Logic
   30: MOV(PID.OUT,HMI_PID_Out);
   31: MOV(PID_ProcessVariable,HMI_PID_PV);
   32: MOV(SP_PID_SP,HMI_PID_SP);
   33: MOV(PID.MAXI,HMI_PID_PVMax);
   34: XIC(PID_En)XIC(DO_Energize)OTE(HMI_PID_Enabled);
   35: XIC(ALM)OTE(HMI_Alarmed);
   36: CPT(HMI_CommandedPosition,AO_CommandPosition*Config_Analog_PositionMaxScaled/Config_AO_PositionMaxRaw);
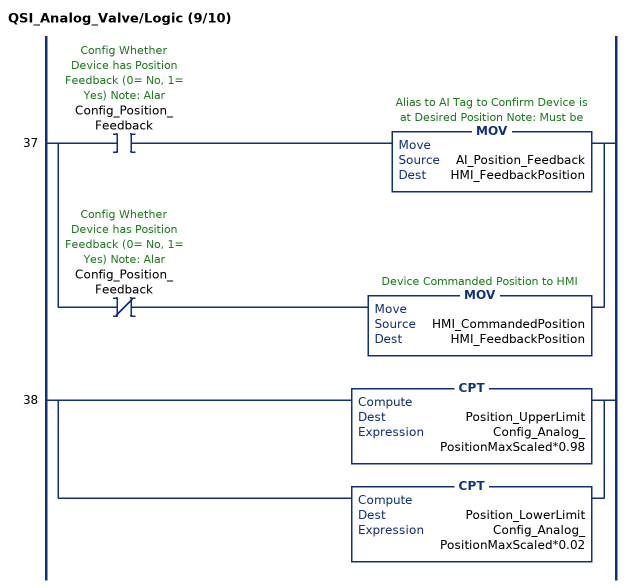
   37: [XIC(Config_Position_Feedback) MOV(AI_Position_Feedback,HMI_FeedbackPosition) ,XIO(Config_Position_Feedback) MOV(HMI_CommandedPosition,HMI_FeedbackPosition) ];
   38: [CPT(Position_UpperLimit,Config_Analog_PositionMaxScaled*0.98) ,CPT(Position_LowerLimit,Config_Analog_PositionMaxScaled*0.02) ];
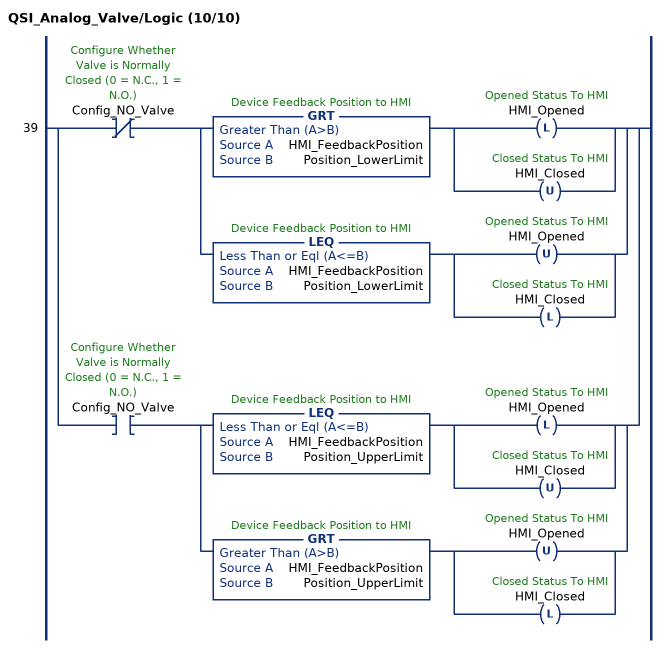
   39: [XIO(Config_NO_Valve) [GRT(HMI_FeedbackPosition,Position_LowerLimit) [OTL(HMI_Opened) ,OTU(HMI_Closed) ] ,LEQ(HMI_FeedbackPosition,Position_LowerLimit) [OTU(HMI_Opened) ,OTL(HMI_Closed) ] ] ,XIC(Config_NO_Valve) [LEQ(HMI_FeedbackPosition,Position_UpperLimit) [OTL(HMI_Opened) ,OTU(HMI_Closed) ] ,GRT(HMI_FeedbackPosition,Position_UpperLimit) [OTU(HMI_Opened) ,OTL(HMI_Closed) ] ] ];
END_ROUTINE
END_ADD_ON_INSTRUCTION
